// TIA Portal project "Bol2" (V17)

(* hardware
DEVICE "S7-1200 station_1"  S7-1200 Station
   slot 0: "Rack_0"  S7-1200 Rack  Rack  V1.0
   slot 1: "PLC_1"  CPU 1214C AC/DC/Rly  6ES7 214-1BG40-0XB0  V4.5
*)

// ===== PLC "PLC_1"  CPU 1214C AC/DC/Rly =====

DATA_BLOCK "Ej1_Datos"   // DB1
{ S7_Optimized_Access := 'TRUE' }
VERSION : 0.1
   VAR
      I : Array[0..4] of Bool;
      "M" : Array[0..1] of Bool;
      Q : Array[0..2] of Bool;
   END_VAR
BEGIN
END_DATA_BLOCK

DATA_BLOCK "Ej2_Datos"   // DB2
{ S7_Optimized_Access := 'TRUE' }
VERSION : 0.1
   VAR
      I : Array[0..4] of Bool;
      Q : Array[0..5] of Bool;
      "M" : Array[0..5] of Bool;
   END_VAR
BEGIN
END_DATA_BLOCK

DATA_BLOCK "Ej3_Datos"   // DB3
{ S7_Optimized_Access := 'TRUE' }
VERSION : 0.1
   VAR
      Sensores : Array[0..2] of Bool;
      Puerta : Bool;
   END_VAR
BEGIN
END_DATA_BLOCK

DATA_BLOCK "Ej4_Datos"   // DB4
{ S7_Optimized_Access := 'TRUE' }
VERSION : 0.1
   VAR
      I : Array[0..1] of Bool;
      Q : Array[0..2] of Bool;
      Cond : Array[0..1] of Int;
   END_VAR
BEGIN
   Cond[0] := 10;
END_DATA_BLOCK

DATA_BLOCK "Ej5_Datos"   // DB5
{ S7_Optimized_Access := 'TRUE' }
VERSION : 0.1
   VAR
      "M" : Array[0..3] of Bool;
      I : Array[0..1] of Bool;
      Rojo : Bool;
      Ambar : Bool;
      Verde : Bool;
   END_VAR
BEGIN
END_DATA_BLOCK

// folder: System blocks/Program resources

DATA_BLOCK "Timer2"   // DB6
{ S7_Optimized_Access := 'TRUE' }
AUTHOR : Simatic
FAMILY : IEC
NAME : IEC_TMR
VERSION : 1.0
// stored: InstanceOfName IEC_TIMER
"IEC_TIMER"
BEGIN
END_DATA_BLOCK

DATA_BLOCK "Timer3"   // DB7
{ S7_Optimized_Access := 'TRUE' }
AUTHOR : Simatic
FAMILY : IEC
NAME : IEC_TMR
VERSION : 1.0
// stored: InstanceOfName IEC_TIMER
"IEC_TIMER"
BEGIN
END_DATA_BLOCK

DATA_BLOCK "Timer1"   // DB8
{ S7_Optimized_Access := 'TRUE' }
AUTHOR : Simatic
FAMILY : IEC
NAME : IEC_TMR
VERSION : 1.0
// stored: InstanceOfName IEC_TIMER
"IEC_TIMER"
BEGIN
END_DATA_BLOCK

DATA_BLOCK "Timer4"   // DB9
{ S7_Optimized_Access := 'TRUE' }
AUTHOR : Simatic
FAMILY : IEC
NAME : IEC_TMR
VERSION : 1.0
// stored: InstanceOfName IEC_TIMER
"IEC_TIMER"
BEGIN
END_DATA_BLOCK

// folder: (top level)

ORGANIZATION_BLOCK "Ej1"   // OB1, LAD, ProgramCycle
TITLE = "Main Program Sweep (Cycle)"
{ S7_Optimized_Access := 'TRUE' }
VERSION : 0.1
   VAR_INPUT
      Initial_Call : Bool;   // Initial call of this OB
      Remanence : Bool;   // =True, if remanent data are available
   END_VAR
BEGIN

REGION Network 1
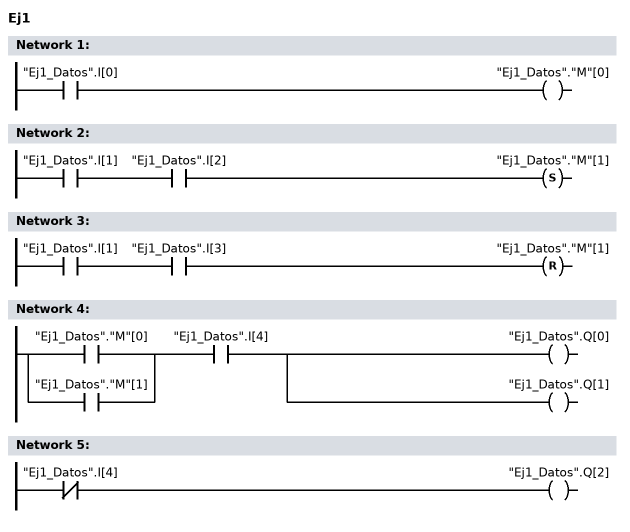
   RUNG wire#powerrail
      Contact( "Ej1_Datos".I[0] )
      Coil( "Ej1_Datos"."M"[0] )
   END_RUNG
   // the same network as SCL:
   "Ej1_Datos"."M"[0] := "Ej1_Datos".I[0];
END_REGION

REGION Network 2
   RUNG wire#powerrail
      Contact( "Ej1_Datos".I[1] )
      Contact( "Ej1_Datos".I[2] )
      S_Coil( "Ej1_Datos"."M"[1] )
   END_RUNG
   // the same network as SCL:
   IF "Ej1_Datos".I[1] AND "Ej1_Datos".I[2] THEN "Ej1_Datos"."M"[1] := TRUE; END_IF;
END_REGION

REGION Network 3
   RUNG wire#powerrail
      Contact( "Ej1_Datos".I[1] )
      Contact( "Ej1_Datos".I[3] )
      R_Coil( "Ej1_Datos"."M"[1] )
   END_RUNG
   // the same network as SCL:
   IF "Ej1_Datos".I[1] AND "Ej1_Datos".I[3] THEN "Ej1_Datos"."M"[1] := FALSE; END_IF;
END_REGION

REGION Network 4
   RUNG wire#powerrail
      Contact( "Ej1_Datos"."M"[0] )
      wire#w1
      Contact( "Ej1_Datos".I[4] )
      wire#w2
      Coil( "Ej1_Datos".Q[0] )
   END_RUNG
   RUNG wire#powerrail
      Contact( "Ej1_Datos"."M"[1] )
   END_RUNG wire#w1
   RUNG wire#w2
      Coil( "Ej1_Datos".Q[1] )
   END_RUNG
   // the same network as SCL:
   "Ej1_Datos".Q[0] := ("Ej1_Datos"."M"[0] OR "Ej1_Datos"."M"[1]) AND "Ej1_Datos".I[4];
   "Ej1_Datos".Q[1] := ("Ej1_Datos"."M"[0] OR "Ej1_Datos"."M"[1]) AND "Ej1_Datos".I[4];
END_REGION

REGION Network 5
   RUNG wire#powerrail
      I_Contact( "Ej1_Datos".I[4] )
      Coil( "Ej1_Datos".Q[2] )
   END_RUNG
   // the same network as SCL:
   "Ej1_Datos".Q[2] := NOT "Ej1_Datos".I[4];
END_REGION
END_ORGANIZATION_BLOCK

ORGANIZATION_BLOCK "Ej2"   // OB123, LAD, ProgramCycle
TITLE = "Main Program Sweep (Cycle)"
{ S7_Optimized_Access := 'TRUE' }
VERSION : 0.1
   VAR_INPUT
      Initial_Call : Bool;   // Initial call of this OB
      Remanence : Bool;   // =True, if remanent data are available
   END_VAR
   VAR_TEMP   // added for the SCL form of the ladder/FBD networks
      _w1 : Bool;
      _w2 : Bool;
   END_VAR
BEGIN

REGION Network 1
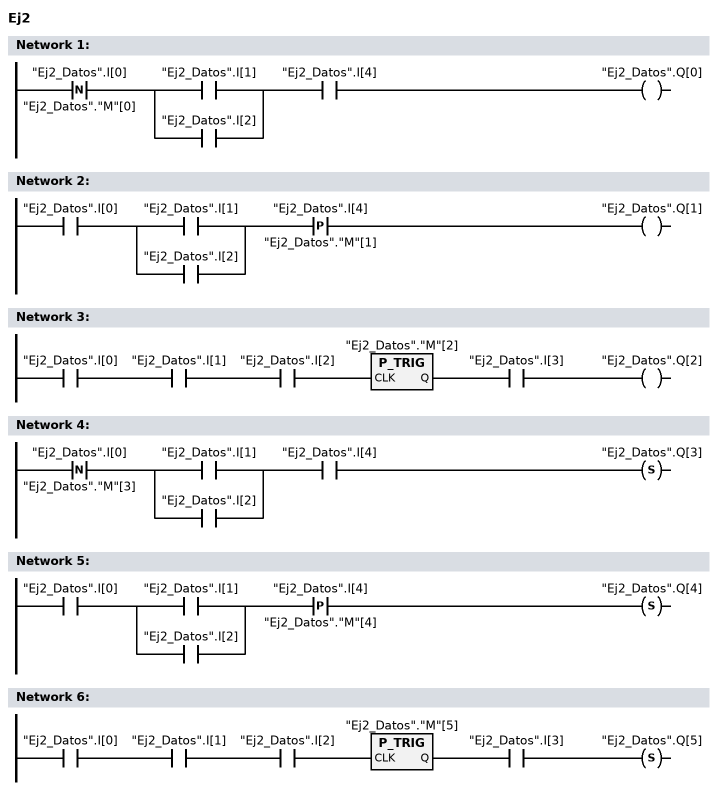
   RUNG wire#powerrail
      N_Contact(operand := "Ej2_Datos".I[0], bit := "Ej2_Datos"."M"[0])
      wire#w1
      Contact( "Ej2_Datos".I[1] )
      wire#w2
      Contact( "Ej2_Datos".I[4] )
      Coil( "Ej2_Datos".Q[0] )
   END_RUNG
   RUNG wire#w1
      Contact( "Ej2_Datos".I[2] )
   END_RUNG wire#w2
   // the same network as SCL:
   #_w1 := NOT "Ej2_Datos".I[0] AND "Ej2_Datos"."M"[0];   // falling edge of "Ej2_Datos".I[0]
   "Ej2_Datos"."M"[0] := "Ej2_Datos".I[0];
   "Ej2_Datos".Q[0] := #_w1 AND ("Ej2_Datos".I[1] OR "Ej2_Datos".I[2]) AND "Ej2_Datos".I[4];
END_REGION

REGION Network 2
   RUNG wire#powerrail
      Contact( "Ej2_Datos".I[0] )
      wire#w1
      Contact( "Ej2_Datos".I[1] )
      wire#w2
      P_Contact(operand := "Ej2_Datos".I[4], bit := "Ej2_Datos"."M"[1])
      Coil( "Ej2_Datos".Q[1] )
   END_RUNG
   RUNG wire#w1
      Contact( "Ej2_Datos".I[2] )
   END_RUNG wire#w2
   // the same network as SCL:
   #_w1 := "Ej2_Datos".I[0] AND ("Ej2_Datos".I[1] OR "Ej2_Datos".I[2]) AND "Ej2_Datos".I[4] AND NOT "Ej2_Datos"."M"[1];   // rising edge of "Ej2_Datos".I[4]
   "Ej2_Datos"."M"[1] := "Ej2_Datos".I[4];
   "Ej2_Datos".Q[1] := #_w1;
END_REGION

REGION Network 3
   RUNG wire#powerrail
      Contact( "Ej2_Datos".I[0] )
      Contact( "Ej2_Datos".I[1] )
      Contact( "Ej2_Datos".I[2] )
      P_Trig( "Ej2_Datos"."M"[2] )
      Contact( "Ej2_Datos".I[3] )
      Coil( "Ej2_Datos".Q[2] )
   END_RUNG
   // the same network as SCL:
   #_w1 := "Ej2_Datos".I[0] AND "Ej2_Datos".I[1] AND "Ej2_Datos".I[2];
   #_w2 := #_w1 AND NOT "Ej2_Datos"."M"[2];   // rising edge
   "Ej2_Datos"."M"[2] := #_w1;
   "Ej2_Datos".Q[2] := #_w2 AND "Ej2_Datos".I[3];
END_REGION

REGION Network 4
   RUNG wire#powerrail
      N_Contact(operand := "Ej2_Datos".I[0], bit := "Ej2_Datos"."M"[3])
      wire#w1
      Contact( "Ej2_Datos".I[1] )
      wire#w2
      Contact( "Ej2_Datos".I[4] )
      S_Coil( "Ej2_Datos".Q[3] )
   END_RUNG
   RUNG wire#w1
      Contact( "Ej2_Datos".I[2] )
   END_RUNG wire#w2
   // the same network as SCL:
   #_w1 := NOT "Ej2_Datos".I[0] AND "Ej2_Datos"."M"[3];   // falling edge of "Ej2_Datos".I[0]
   "Ej2_Datos"."M"[3] := "Ej2_Datos".I[0];
   IF #_w1 AND ("Ej2_Datos".I[1] OR "Ej2_Datos".I[2]) AND "Ej2_Datos".I[4] THEN
       "Ej2_Datos".Q[3] := TRUE;
   END_IF;
END_REGION

REGION Network 5
   RUNG wire#powerrail
      Contact( "Ej2_Datos".I[0] )
      wire#w1
      Contact( "Ej2_Datos".I[1] )
      wire#w2
      P_Contact(operand := "Ej2_Datos".I[4], bit := "Ej2_Datos"."M"[4])
      S_Coil( "Ej2_Datos".Q[4] )
   END_RUNG
   RUNG wire#w1
      Contact( "Ej2_Datos".I[2] )
   END_RUNG wire#w2
   // the same network as SCL:
   #_w1 := "Ej2_Datos".I[0] AND ("Ej2_Datos".I[1] OR "Ej2_Datos".I[2]) AND "Ej2_Datos".I[4] AND NOT "Ej2_Datos"."M"[4];   // rising edge of "Ej2_Datos".I[4]
   "Ej2_Datos"."M"[4] := "Ej2_Datos".I[4];
   IF #_w1 THEN "Ej2_Datos".Q[4] := TRUE; END_IF;
END_REGION

REGION Network 6
   RUNG wire#powerrail
      Contact( "Ej2_Datos".I[0] )
      Contact( "Ej2_Datos".I[1] )
      Contact( "Ej2_Datos".I[2] )
      P_Trig( "Ej2_Datos"."M"[5] )
      Contact( "Ej2_Datos".I[3] )
      S_Coil( "Ej2_Datos".Q[5] )
   END_RUNG
   // the same network as SCL:
   #_w1 := "Ej2_Datos".I[0] AND "Ej2_Datos".I[1] AND "Ej2_Datos".I[2];
   #_w2 := #_w1 AND NOT "Ej2_Datos"."M"[5];   // rising edge
   "Ej2_Datos"."M"[5] := #_w1;
   IF #_w2 AND "Ej2_Datos".I[3] THEN "Ej2_Datos".Q[5] := TRUE; END_IF;
END_REGION
END_ORGANIZATION_BLOCK

ORGANIZATION_BLOCK "Ej3"   // OB124, LAD, ProgramCycle
TITLE = "Main Program Sweep (Cycle)"
{ S7_Optimized_Access := 'TRUE' }
VERSION : 0.1
   VAR_INPUT
      Initial_Call : Bool;   // Initial call of this OB
      Remanence : Bool;   // =True, if remanent data are available
   END_VAR
BEGIN

REGION Network 1
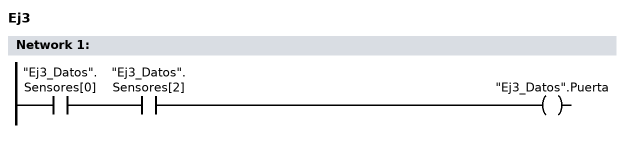
   RUNG wire#powerrail
      Contact( "Ej3_Datos".Sensores[0] )
      Contact( "Ej3_Datos".Sensores[2] )
      Coil( "Ej3_Datos".Puerta )
   END_RUNG
   // the same network as SCL:
   "Ej3_Datos".Puerta := "Ej3_Datos".Sensores[0] AND "Ej3_Datos".Sensores[2];
END_REGION
END_ORGANIZATION_BLOCK

ORGANIZATION_BLOCK "Ej4"   // OB125, LAD, ProgramCycle
TITLE = "Main Program Sweep (Cycle)"
{ S7_Optimized_Access := 'TRUE' }
VERSION : 0.1
   VAR_INPUT
      Initial_Call : Bool;   // Initial call of this OB
      Remanence : Bool;   // =True, if remanent data are available
   END_VAR
   VAR_TEMP   // added for the SCL form of the ladder/FBD networks
      _w1 : Bool;
   END_VAR
BEGIN

REGION Network 1
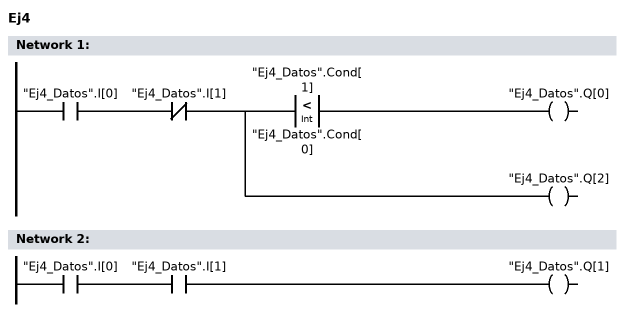
   RUNG wire#powerrail
      Contact( "Ej4_Datos".I[0] )
      I_Contact( "Ej4_Datos".I[1] )
      wire#w1
      { S7_Templates := "SrcType := Int" } LT_Contact(in1 := "Ej4_Datos".Cond[1], in2 := "Ej4_Datos".Cond[0])
      Coil( "Ej4_Datos".Q[0] )
   END_RUNG
   RUNG wire#w1
      Coil( "Ej4_Datos".Q[2] )
   END_RUNG
   // the same network as SCL:
   #_w1 := "Ej4_Datos".I[0] AND NOT "Ej4_Datos".I[1];
   "Ej4_Datos".Q[0] := #_w1 AND ("Ej4_Datos".Cond[1] < "Ej4_Datos".Cond[0]);
   "Ej4_Datos".Q[2] := #_w1;
END_REGION

REGION Network 2
   RUNG wire#powerrail
      Contact( "Ej4_Datos".I[0] )
      Contact( "Ej4_Datos".I[1] )
      Coil( "Ej4_Datos".Q[1] )
   END_RUNG
   // the same network as SCL:
   "Ej4_Datos".Q[1] := "Ej4_Datos".I[0] AND "Ej4_Datos".I[1];
END_REGION
END_ORGANIZATION_BLOCK

ORGANIZATION_BLOCK "Ej5"   // OB126, LAD, ProgramCycle
TITLE = "Main Program Sweep (Cycle)"
{ S7_Optimized_Access := 'TRUE' }
VERSION : 0.1
   VAR_INPUT
      Initial_Call : Bool;   // Initial call of this OB
      Remanence : Bool;   // =True, if remanent data are available
   END_VAR
   VAR_TEMP   // added for the SCL form of the ladder/FBD networks
      _w1 : Bool;
      _w2 : Bool;
   END_VAR
BEGIN

REGION Network 1
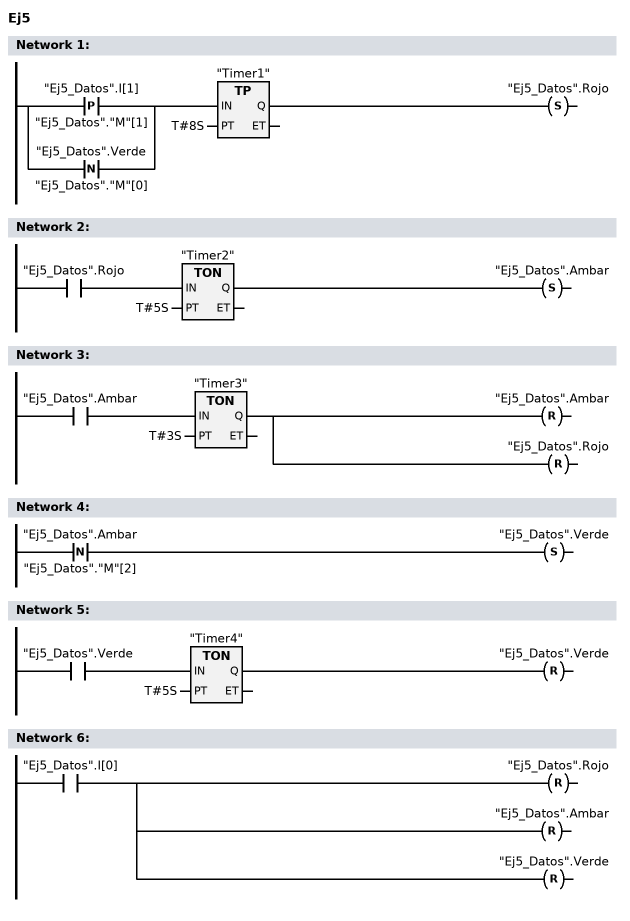
   #_w1 := "Ej5_Datos".I[1] AND NOT "Ej5_Datos"."M"[1];   // rising edge of "Ej5_Datos".I[1]
   "Ej5_Datos"."M"[1] := "Ej5_Datos".I[1];
   #_w2 := NOT "Ej5_Datos".Verde AND "Ej5_Datos"."M"[0];   // falling edge of "Ej5_Datos".Verde
   "Ej5_Datos"."M"[0] := "Ej5_Datos".Verde;
   "Timer1".TP(IN := #_w1 OR #_w2, PT := T#8S);
   IF "Timer1".Q THEN "Ej5_Datos".Rojo := TRUE; END_IF;
END_REGION

REGION Network 2
   "Timer2".TON(IN := "Ej5_Datos".Rojo, PT := T#5S);
   IF "Timer2".Q THEN "Ej5_Datos".Ambar := TRUE; END_IF;
END_REGION

REGION Network 3
   "Timer3".TON(IN := "Ej5_Datos".Ambar, PT := T#3S);
   IF "Timer3".Q THEN
       "Ej5_Datos".Ambar := FALSE;
       "Ej5_Datos".Rojo := FALSE;
   END_IF;
END_REGION

REGION Network 4
   RUNG wire#powerrail
      N_Contact(operand := "Ej5_Datos".Ambar, bit := "Ej5_Datos"."M"[2])
      S_Coil( "Ej5_Datos".Verde )
   END_RUNG
   // the same network as SCL:
   #_w1 := NOT "Ej5_Datos".Ambar AND "Ej5_Datos"."M"[2];   // falling edge of "Ej5_Datos".Ambar
   "Ej5_Datos"."M"[2] := "Ej5_Datos".Ambar;
   IF #_w1 THEN "Ej5_Datos".Verde := TRUE; END_IF;
END_REGION

REGION Network 5
   "Timer4".TON(IN := "Ej5_Datos".Verde, PT := T#5S);
   IF "Timer4".Q THEN "Ej5_Datos".Verde := FALSE; END_IF;
END_REGION

REGION Network 6
   RUNG wire#powerrail
      Contact( "Ej5_Datos".I[0] )
      wire#w1
      R_Coil( "Ej5_Datos".Rojo )
   END_RUNG
   RUNG wire#w1
      R_Coil( "Ej5_Datos".Ambar )
   END_RUNG
   RUNG wire#w1
      R_Coil( "Ej5_Datos".Verde )
   END_RUNG
   // the same network as SCL:
   IF "Ej5_Datos".I[0] THEN
       "Ej5_Datos".Rojo := FALSE;
       "Ej5_Datos".Ambar := FALSE;
       "Ej5_Datos".Verde := FALSE;
   END_IF;
END_REGION
END_ORGANIZATION_BLOCK